# EPICS StreamDevice protocol: epics/protocols/gain_mux.proto
Terminator = LF;
ExtraInput = Ignore;
ReplyTimeout = 2500;

write_mux {
	out "sc32_set_gain \$1 0x%04x";
	in;
}
